// TwinCAT 3 PLC project tectrl
// ProgramVersion: 3.1.0.8
// libraries:
//   Tc2_Standard, * (Beckhoff Automation GmbH)
//   Tc2_System, * (Beckhoff Automation GmbH)
//   Tc3_Interfaces, * (Beckhoff Automation GmbH)
//   Tc3_Module, * (Beckhoff Automation GmbH)
//   Tc2_ControllerToolbox,3.4.1.0,Beckhoff Automation GmbH
//   Tc2_Math,3.3.0.0,Beckhoff Automation GmbH
//   Tc2_Utilities,3.3.8.0,Beckhoff Automation GmbH
//   Tc3_CM,newest,Beckhoff Automation GmbH
//   Tc3_MemMan,3.3.1.0,Beckhoff Automation GmbH
// project tree:
//   GVLs/ GVL.TcGVL
//   / PlcTask.TcTTO
//   POUs/components/ fb_ac_measurements.TcPOU, fb_discrete_pi.TcPOU, fb_flow_rate.TcPOU, fb_prod_feedforward.TcPOU, fb_ratio_trimming.TcPOU, fb_slewrate_limiter.TcPOU, fb_vel_pi.TcPOU (not stored), fb_xmeas_acquire.TcPOU (not stored), fb_unitdelay_real.TcPOU (not stored)
//   POUs/debug/ fb_generate_random_value.TcPOU (not stored), fb_xmeas_simulated.TcPOU (not stored)
//   POUs/ ldrMain.TcPOU
//   POUs/subsystems/ fb_ac_ratio_ctrl.TcPOU, fb_level_ctrl.TcPOU, fb_prod_rate_ctrl.TcPOU, fb_prod_comp_ctrl.TcPOU, fb_feed_ratio_ctrl.TcPOU (not stored), fb_temp_ctrl.TcPOU
//   POUs/test/ fb_test_xmeas_simulated.TcPOU (not stored)
// real-time tasks:
//   TASK PlcTask: cycle T#100000us, priority 20, ADS port 350

CONFIGURATION tectrl
    RESOURCE PLC ON TwinCAT3
        TASK PlcTask(INTERVAL := T#100000us, PRIORITY := 20);
        PROGRAM ldrMain WITH PlcTask : ldrMain;
    END_RESOURCE
END_CONFIGURATION

// ---- GVLs/GVL.TcGVL
VAR_GLOBAL
	
	// used for main start/stop/estop
	g_RUNNING: BOOL;
	g_START: BOOL;
	
	// E-STOP
	g_ESTOP: BOOL := TRUE;
	
	// loop control constants
	g_Ts_base : REAL := 0.001;
	g_Ts : REAL := 0.1;
	
	// the initial setpoints
	g_set_production: 		REAL := 22.89;
	g_set_stip_level: 		REAL := 50;
	g_set_sep_level:  		REAL := 50;
	g_set_reactor_level: 	REAL := 65;
	g_set_reactor_press: 	REAL := 2800;
	g_set_mol_pct_g:	 	REAL := 53.8;
	g_set_ya:				REAL := 100*32.2/(32.2+18.8);
	g_set_yac:				REAL := 32.2+18.8;
	g_set_reactor_temp:		REAL := 122.9;
	g_set_rcycle_valve_pos: REAL := 0;
	g_set_steam_valve_pos:	REAL := 0;
	g_set_agitator_speed:	REAL :=	100;		
	g_set_separator_temp:	REAL := SP17_0;
	
	// storage variables for sub-controllers
	g_xmeas: ARRAY [1..41] 	OF REAL;
	g_xmv: ARRAY [1..12] 	OF REAL := [50,50,65,2800,22.89,63.1373,51,122.9,0,0,100,53.8];
	g_rx: ARRAY [1..7] 		OF REAL;
	
	// production rate variables
	g_Prodsp: REAL;
	g_Fp: REAL;
	
	// Percent G Composition
	g_PctGsp: REAL;
	g_Eadj: REAL :=1.0;
	
	
	
END_VAR

VAR_GLOBAL CONSTANT
	Fp_0: REAL :=100;
	r_0 : ARRAY [1..7] OF REAL := 
		[0.251/Fp_0, 3664/Fp_0, 4509/Fp_0, 9.35/Fp_0, 0.337/Fp_0, 25.16/Fp_0, 22.95/Fp_0];    
              		
	xmv_0 : ARRAY [1..12] OF REAL := 
		[50,50,65,2800,22.89,63.1373,51,122.9,0,0,100,53.8];
	
	SP17_0 : REAL := 0.0;  // need value !!!
	Eadj_0 : REAL := 0.0;  // need value !!!
	ProdspGain: REAL := 100/22.89;	
END_VAR

// ---- POUs/ldrMain.TcPOU
PROGRAM ldrMain


// Notes
//  I imagine that the control loops can run as independent threads/tasks under the main PlcTask
//  xmeas, xmv, r, and maybe others could be stored in a GVL 
VAR
	
	// data acquitistion from IO blocks
	xmeas_acquire: fb_xmeas_acquire;

	// Molar Percent G control loop
	//pct_g_dpi: fb_discrete_pi		  := (kc:=1, ti:=0.001/60, Ts:=g_Ts_base, hi :=100, lo:=0, x0:=Eadj_0);
	
	// production rate control loop
	prod_rate_loop: fb_prod_rate_ctrl := (kc:=3.2, ti:=120/60, ts:=g_Ts_base, x0:=0, hi:=30, lo:=0);	
	
	// feed ratio control loop
	feed_ratio_ctrl: fb_feed_ratio_ctrl;
	
	// process levels/invetory controller
	level_ctrl: fb_level_ctrl;
		
	// product comnposition controller
	prod_comp_ctrl: fb_prod_comp_ctrl;
	
	// A & C ratio controller
	ac_ratio_ctrl: fb_ac_ratio_ctrl;
	
	// temperature controller
	temp_ctrl: fb_temp_ctrl;
	
END_VAR

VAR_INPUT
	
END_VAR
VAR // added by the converter: edge detectors and wires of the graphical bodies
    _w1 : BOOL;
END_VAR

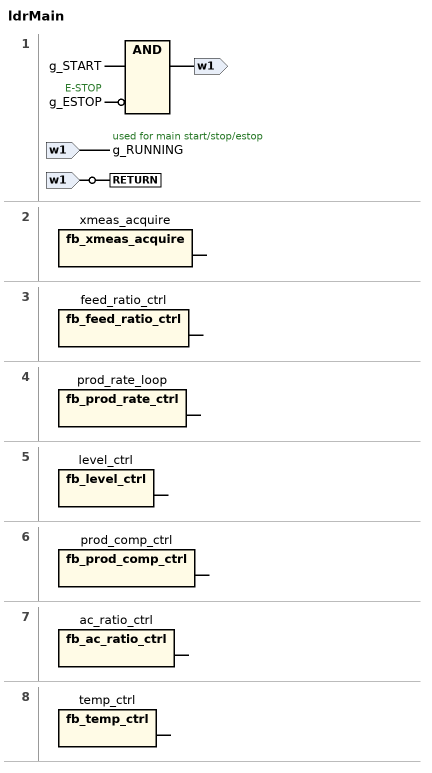
// NETWORK 1
//   g_ESTOP: E-STOP
//   g_RUNNING: used for main start/stop/estop
_w1 := g_START AND NOT g_ESTOP;
g_RUNNING := _w1;
IF NOT _w1 THEN RETURN; END_IF

// NETWORK 2
//   xmeas_acquire: data acquitistion from IO blocks
xmeas_acquire(); // fb_xmeas_acquire

// NETWORK 3
//   feed_ratio_ctrl: feed ratio control loop
feed_ratio_ctrl(); // fb_feed_ratio_ctrl

// NETWORK 4
//   prod_rate_loop: production rate control loop
prod_rate_loop(); // fb_prod_rate_ctrl

// NETWORK 5
//   level_ctrl: process levels/invetory controller
level_ctrl(); // fb_level_ctrl

// NETWORK 6
//   prod_comp_ctrl: product comnposition controller
prod_comp_ctrl(); // fb_prod_comp_ctrl

// NETWORK 7
//   ac_ratio_ctrl: A & C ratio controller
ac_ratio_ctrl(); // fb_ac_ratio_ctrl

// NETWORK 8
//   temp_ctrl: temperature controller
temp_ctrl(); // fb_temp_ctrl

END_PROGRAM

// ---- POUs/subsystems/fb_prod_rate_ctrl.TcPOU
FUNCTION_BLOCK fb_prod_rate_ctrl

VAR_INPUT
	kc: REAL;
	ti:REAL;
	ts:REAL;
	hi:REAL;
	lo:REAL;
	x0:REAL := 0;
	set_prod_rate: REAL := g_set_production;
	//xmv17: REAL;

END_VAR

VAR_OUTPUT
	Prodsp: REAL := 0;
	Fp: REAL :=0;
END_VAR

VAR
	
	vel_p: fb_vel_pi;
	x: FB_CTRL_2POINT;
	zoh_real_0: fb_zoh_real := (xlast := x0 );
	change_rate_limit: FB_CTRL_LIMITER := (stInternalParams := (fMinOutput := -0.286875, fMaxOutput := 0.286875));
	rate: REAL := 0;
	
	prodsp_scaled: REAL;
	calc_change_rate: FB_CTRL_D;
	integrate_change_rate: FB_CTRL_I;
	prod_rate_saturate: FB_CTRL_LIMITER;
	prod_rate_saturate_params: ST_CTRL_LIMITER_PARAMS := (fMinOutput := lo, fMaxOutput := hi);
	last_prod_rate: REAL := 0.0;
	
	stparams_calc_change_rate: ST_CTRL_D_PARAMS;
	stparams_change_rate_limit: ST_CTRL_LIMITER_PARAMS;
	stparams_integrate_change_rate: ST_CTRL_I_PARAMS;
	
END_VAR

VAR CONSTANT
	ProdspGain: REAL := 100/22.89;
END_VAR

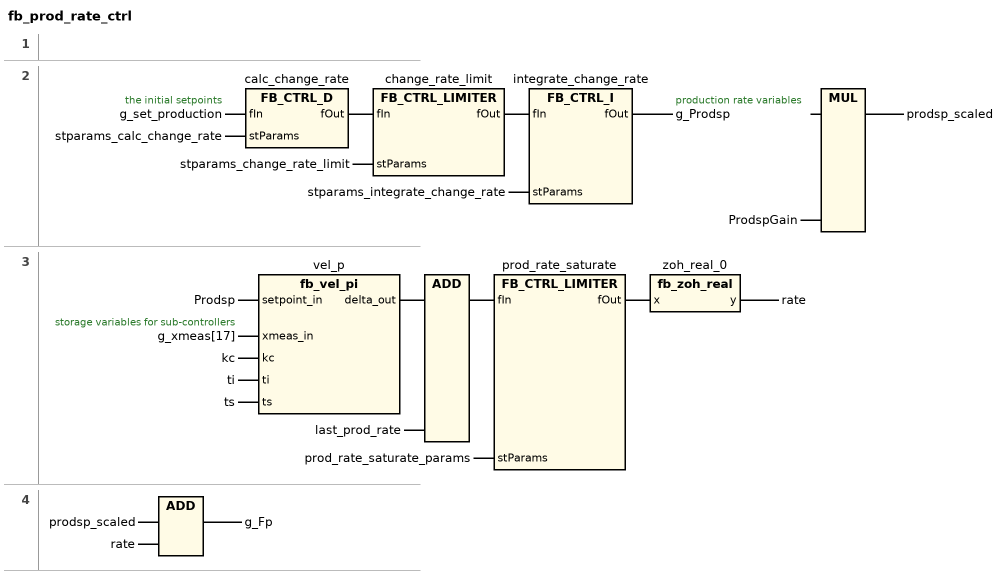
// NETWORK 1

// NETWORK 2
//   g_set_production: the initial setpoints
//   g_Prodsp: production rate variables
calc_change_rate(fIn := g_set_production, stParams := stparams_calc_change_rate); // FB_CTRL_D
change_rate_limit(fIn := calc_change_rate.fOut, stParams := stparams_change_rate_limit); // FB_CTRL_LIMITER
integrate_change_rate(fIn := change_rate_limit.fOut, stParams := stparams_integrate_change_rate); // FB_CTRL_I
g_Prodsp := integrate_change_rate.fOut;
prodsp_scaled := integrate_change_rate.fOut * ProdspGain;

// NETWORK 3
//   g_xmeas[17]: storage variables for sub-controllers
vel_p(setpoint_in := Prodsp, xmeas_in := g_xmeas[17], kc := kc, ti := ti, ts := ts); // fb_vel_pi
prod_rate_saturate(fIn := vel_p.delta_out + last_prod_rate, stParams := prod_rate_saturate_params); // FB_CTRL_LIMITER
zoh_real_0(x := prod_rate_saturate.fOut); // fb_zoh_real
rate := zoh_real_0.y;

// NETWORK 4
g_Fp := prodsp_scaled + rate;

END_FUNCTION_BLOCK

// ---- POUs/subsystems/fb_level_ctrl.TcPOU
FUNCTION_BLOCK fb_level_ctrl

VAR_INPUT
END_VAR

VAR_OUTPUT
END_VAR

VAR
	stripper_level_dpi: fb_discrete_pi			:= (kc:=2E-4, ti:=200/60, Ts:=g_Ts_base, hi :=100, lo:=0, x0:=r_0[7]);
	separator_level_dpi: fb_discrete_pi			:= (kc:=-1E-3, ti:=200/60, Ts:=g_Ts_base, hi :=100, lo:=0, x0:=r_0[6]);
	reactor_level_dpi: fb_discrete_pi			:= (kc:=0.8, ti:=60/60, Ts:=g_Ts_base, hi :=100, lo:=0, x0:=SP17_0);
	reactor_pressure_dpi: fb_discrete_pi		:= (kc:=-1E-4, ti:=20/60, Ts:=g_Ts_base, hi :=100, lo:=0, x0:=r_0[5]);
	reactor_temp_dpi: fb_discrete_pi			:= (kc:=-8, ti:=7.5/60, Ts:=g_Ts_base, hi :=100, lo:=0, x0:=xmv_0[10]);		
END_VAR

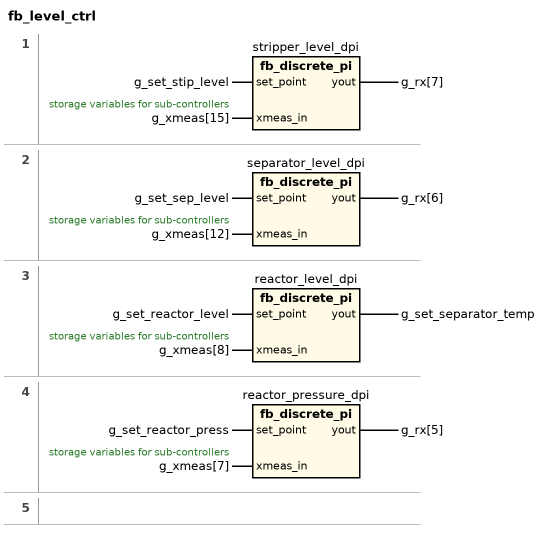
// NETWORK 1
//   g_xmeas[15]: storage variables for sub-controllers
stripper_level_dpi(set_point := g_set_stip_level, xmeas_in := g_xmeas[15]); // fb_discrete_pi
g_rx[7] := stripper_level_dpi.yout;

// NETWORK 2
//   g_xmeas[12]: storage variables for sub-controllers
separator_level_dpi(set_point := g_set_sep_level, xmeas_in := g_xmeas[12]); // fb_discrete_pi
g_rx[6] := separator_level_dpi.yout;

// NETWORK 3
//   g_xmeas[8]: storage variables for sub-controllers
reactor_level_dpi(set_point := g_set_reactor_level, xmeas_in := g_xmeas[8]); // fb_discrete_pi
g_set_separator_temp := reactor_level_dpi.yout;

// NETWORK 4
//   g_xmeas[7]: storage variables for sub-controllers
reactor_pressure_dpi(set_point := g_set_reactor_press, xmeas_in := g_xmeas[7]); // fb_discrete_pi
g_rx[5] := reactor_pressure_dpi.yout;

// NETWORK 5

END_FUNCTION_BLOCK

// ---- POUs/components/fb_discrete_pi.TcPOU
FUNCTION_BLOCK fb_discrete_pi

VAR_INPUT
	// signal inputs
	set_point: REAL := 0.0;
	xmeas_in: REAL := 0.0;
	
	// parameters
	kc: REAL;
	ti: REAL;
	ts: REAL;
	hi: REAL := 100;
	lo: REAL;
	x0: REAL;
		
END_VAR

VAR_OUTPUT
	yout: REAL; // needs to be initialized by caller
END_VAR

VAR
	vel_pi: fb_vel_pi := (kc:=kc, ti:=ti, ts:=ts);
	dpi_unit_delay: fb_unitdelay_real := (xlast:=x0);
END_VAR

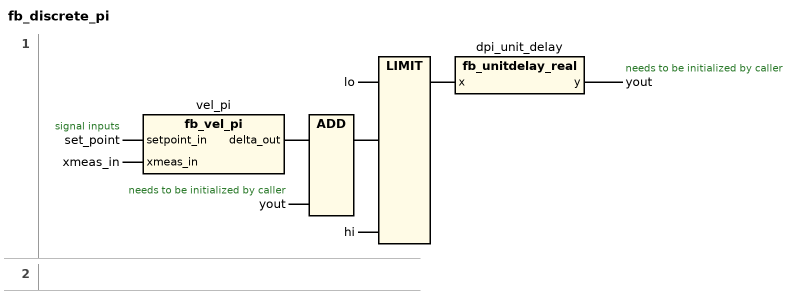
// NETWORK 1
//   set_point: signal inputs
//   yout: needs to be initialized by caller
vel_pi(setpoint_in := set_point, xmeas_in := xmeas_in); // fb_vel_pi
dpi_unit_delay(x := LIMIT(lo, vel_pi.delta_out + yout, hi)); // fb_unitdelay_real
yout := dpi_unit_delay.y;

// NETWORK 2

END_FUNCTION_BLOCK

// ---- POUs/subsystems/fb_prod_comp_ctrl.TcPOU
FUNCTION_BLOCK fb_prod_comp_ctrl

VAR_INPUT
	kc: REAL := 0.0;
	ti:REAL := 0.0;
	ts:REAL := 0.0;
	hi:REAL := 0.0;
	lo:REAL := 0.0;
	x0:REAL := 0.0;
	set_prod_rate: REAL := g_set_production;
	//xmv17: REAL;

END_VAR

VAR_OUTPUT
	Prodsp: REAL := 0;
	Fp: REAL :=0;
END_VAR

VAR
	
	pct_g_dpi: fb_discrete_pi := (kc := 0.4, ti := 100.0, ts := g_Ts_base, hi := 100, lo:=0.0);
	zoh_real_0: fb_zoh_real := (xlast := x0 );
	change_rate_limit: FB_CTRL_LIMITER := (stInternalParams := (fMinOutput := -0.286875, fMaxOutput := 0.286875));
	rate: REAL := 0;
	
	prodsp_scaled: REAL;
	calc_change_rate: FB_CTRL_D;
	integrate_change_rate: FB_CTRL_I;
	prod_rate_saturate: FB_CTRL_LIMITER;
	prod_rate_saturate_params: ST_CTRL_LIMITER_PARAMS := (fMinOutput := lo, fMaxOutput := hi);
	last_prod_rate: REAL := 0.0;
	
	stparams_calc_change_rate: ST_CTRL_D_PARAMS;
	stparams_change_rate_limit: ST_CTRL_LIMITER_PARAMS;
	stparams_integrate_change_rate: ST_CTRL_I_PARAMS;
	
	pctgsp: REAL := 0.0;
	
	
	prod_feedforward: fb_prod_feedforward;
END_VAR

VAR CONSTANT
	ProdspGain: REAL := 100/22.89;
END_VAR

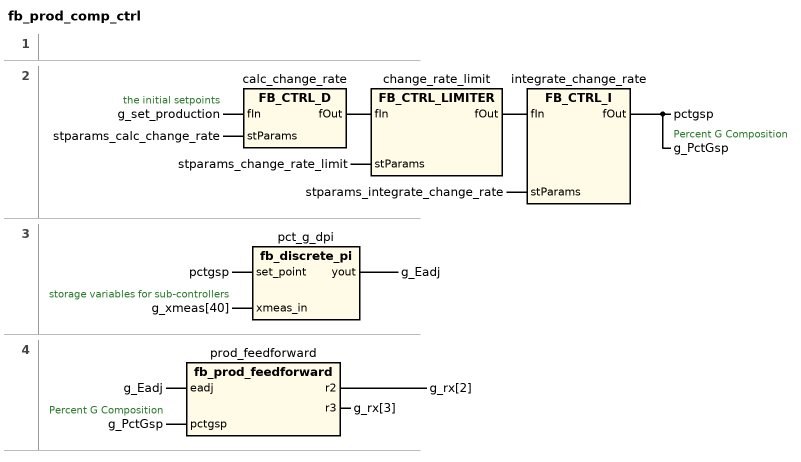
// NETWORK 1

// NETWORK 2
//   g_set_production: the initial setpoints
//   g_PctGsp: Percent G Composition
calc_change_rate(fIn := g_set_production, stParams := stparams_calc_change_rate); // FB_CTRL_D
change_rate_limit(fIn := calc_change_rate.fOut, stParams := stparams_change_rate_limit); // FB_CTRL_LIMITER
integrate_change_rate(fIn := change_rate_limit.fOut, stParams := stparams_integrate_change_rate); // FB_CTRL_I
pctgsp := integrate_change_rate.fOut;
g_PctGsp := integrate_change_rate.fOut;

// NETWORK 3
//   g_xmeas[40]: storage variables for sub-controllers
pct_g_dpi(set_point := pctgsp, xmeas_in := g_xmeas[40]); // fb_discrete_pi
g_Eadj := pct_g_dpi.yout;

// NETWORK 4
//   g_PctGsp: Percent G Composition
prod_feedforward(eadj := g_Eadj, pctgsp := g_PctGsp, r3 => g_rx[3]); // fb_prod_feedforward
g_rx[2] := prod_feedforward.r2;

END_FUNCTION_BLOCK

// ---- POUs/components/fb_prod_feedforward.TcPOU
FUNCTION_BLOCK fb_prod_feedforward

VAR_INPUT	
	eadj: REAL;
	pctgsp: REAL;
END_VAR

VAR_OUTPUT
	r2: REAL;
	r3: REAL;
END_VAR

VAR
	pctgspP2: REAL;
	pctgspP3: REAL;
	eadjProd1: REAL;
	eadjProd2: REAL;
END_VAR

VAR CONSTANT
	P2: ARRAY[0..2] OF REAL := [1.5192E-3, 5.9446E-1, 2.7690E-1]; 
	P3: ARRAY[0..2] OF REAL := [-1.1377E-3, -8.0893E-1, 9.1060E1]; 
END_VAR


pctgspP2 := P2[0]*EXPT(pctgsp,2) + P2[1]*pctgsp + P2[2];
pctgspP3 := P2[0]*EXPT(pctgsp,2) + P2[1]*pctgsp + P2[2];
g_rx[2] :=  pctgspP2 - (32*eadj)/g_Fp;
g_rx[3] :=  pctgspP2 + (46*eadj)/g_Fp;

END_FUNCTION_BLOCK

// ---- POUs/subsystems/fb_ac_ratio_ctrl.TcPOU
FUNCTION_BLOCK fb_ac_ratio_ctrl

VAR_INPUT
	(*
	set_ya:  REAL := g_set_ya;
	set_yac: REAL := g_set_yac;
	xmeas11: REAL := g_xmeas[11];
	xmeas23: REAL := g_xmeas[23];
	xmeas25: REAL := g_xmeas[25];
	*)
END_VAR

VAR_OUTPUT
END_VAR

VAR
	// A & C measurements
	yA: 	REAL;
	yAC:	REAL;
	
	// yA control looop
	ya_control: fb_vel_pi := (kc := 0.0002, ti := 1.0, ts := g_Ts);
	ya_control_kc :	REAL := 0.0;
	loop14:	REAL := 0.0;
	
	// yAC control loop
	yac_control: fb_vel_pi := (kc := 0.0003, ti := 2, ts := g_Ts);
	loop15: REAL := 0.0;	
	
	// ratio trimming
	ratio_trimming: fb_ratio_trimming;
	
	// fine ac adjustments
	ac_measurements: fb_ac_measurements;
	separator_temp_dpi: fb_discrete_pi		:= (kc:=-4, ti:=15/60, Ts:=g_Ts_base, hi :=100, lo:=0, yout:=xmv_0[11]);	
	ratio_trimming_0: fb_ratio_trimming 	:= (r1 := g_rx[1], r4 := g_rx[4]);

END_VAR

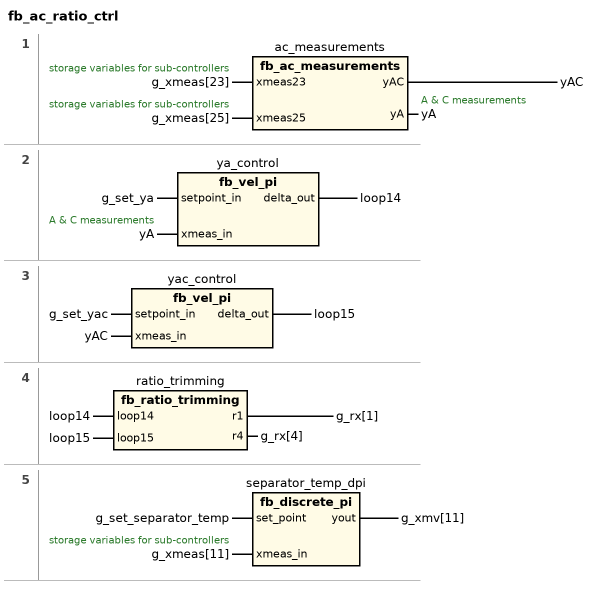
// NETWORK 1
//   ac_measurements: fine ac adjustments
//   g_xmeas[23]: storage variables for sub-controllers
//   g_xmeas[25]: storage variables for sub-controllers
//   yA: A & C measurements
ac_measurements(xmeas23 := g_xmeas[23], xmeas25 := g_xmeas[25], yA => yA); // fb_ac_measurements
yAC := ac_measurements.yAC;

// NETWORK 2
//   ya_control: yA control looop
//   yA: A & C measurements
ya_control(setpoint_in := g_set_ya, xmeas_in := yA); // fb_vel_pi
loop14 := ya_control.delta_out;

// NETWORK 3
//   yac_control: yAC control loop
yac_control(setpoint_in := g_set_yac, xmeas_in := yAC); // fb_vel_pi
loop15 := yac_control.delta_out;

// NETWORK 4
//   ratio_trimming: ratio trimming
ratio_trimming(loop14 := loop14, loop15 := loop15, r4 => g_rx[4]); // fb_ratio_trimming
g_rx[1] := ratio_trimming.r1;

// NETWORK 5
//   g_xmeas[11]: storage variables for sub-controllers
separator_temp_dpi(set_point := g_set_separator_temp, xmeas_in := g_xmeas[11]); // fb_discrete_pi
g_xmv[11] := separator_temp_dpi.yout;

END_FUNCTION_BLOCK

// ---- POUs/components/fb_ratio_trimming.TcPOU
FUNCTION_BLOCK fb_ratio_trimming

VAR_INPUT
	loop14: REAL;
	loop15: REAL;
END_VAR

VAR_OUTPUT
	r1: REAL;
	r4: REAL;
END_VAR

VAR
END_VAR


r1 := loop14 + r1;
r4 := loop15 - loop14 + r4;

END_FUNCTION_BLOCK

// ---- POUs/components/fb_ac_measurements.TcPOU
FUNCTION_BLOCK fb_ac_measurements

VAR_INPUT
	xmeas23 : REAL := 0.0;
	xmeas25 : REAL := 0.0;
END_VAR

VAR_OUTPUT
	yAC : REAL := 0.0;
	yA : REAL := 0.0;
	
	
END_VAR

VAR
END_VAR


yAC := xmeas23 + xmeas25;
yA := xmeas23*100/yAC;

END_FUNCTION_BLOCK

// ---- POUs/subsystems/fb_temp_ctrl.TcPOU
FUNCTION_BLOCK fb_temp_ctrl

VAR_INPUT
END_VAR

VAR_OUTPUT	
END_VAR

VAR
	separator_temp_dpi: fb_discrete_pi		:= (kc:=-4, ti:=15/60, Ts:=g_Ts_base, hi :=100, lo:=0, yout:=xmv_0[11]);	
	reactor_temp_dpi: fb_discrete_pi		:= (kc:=-8, ti:=7.5/60, Ts:=g_Ts_base, hi :=100, lo:=0, yout:=xmv_0[10]);
	
END_VAR

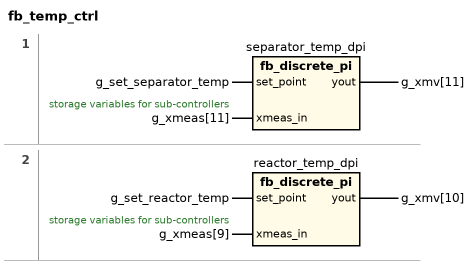
// NETWORK 1
//   g_xmeas[11]: storage variables for sub-controllers
separator_temp_dpi(set_point := g_set_separator_temp, xmeas_in := g_xmeas[11]); // fb_discrete_pi
g_xmv[11] := separator_temp_dpi.yout;

// NETWORK 2
//   g_xmeas[9]: storage variables for sub-controllers
reactor_temp_dpi(set_point := g_set_reactor_temp, xmeas_in := g_xmeas[9]); // fb_discrete_pi
g_xmv[10] := reactor_temp_dpi.yout;

END_FUNCTION_BLOCK

// ---- POUs/components/fb_flow_rate.TcPOU
FUNCTION_BLOCK fb_flow_rate

VAR_INPUT
	// signal inputs
	ratio_in: REAL := 0.0;
	xmeas_in: REAL := 0.0;
	
	// parameters
	kc: REAL := 0.0;
	ti: REAL := 0.0;
	ts: REAL := 0.0;
	hi: REAL := 2E32;
	lo: REAL := 0;
	
END_VAR

VAR_OUTPUT
	yout: REAL; // needs to be initialized by caller
END_VAR

VAR
	vel_pi: fb_vel_pi;
END_VAR

END_FUNCTION_BLOCK

// ---- POUs/components/fb_slewrate_limiter.TcPOU
FUNCTION_BLOCK fb_slewrate_limiter

VAR_INPUT
	in: REAL;
	pos_slewrate_limit: REAL := 0.0;
	neg_slewrate_limit: REAL := 0.0;
END_VAR

VAR_OUTPUT
	out: REAL;
END_VAR

VAR
	
	last_in: REAL := g_set_production;
	slope: REAL;

	fbCTRL_GET_TASK_CYCLETIME   : FB_CTRL_GET_TASK_CYCLETIME;
	tTaskCycleTime: TIME;
	bCycleTimeValid: BOOL;
	eErrorId: TC2_CONTROLLERTOOLBOX.E_CTRL_ERRORCODES;
	bError: BOOL;
    eState: E_CTRL_STATE;

END_VAR


fbCTRL_GET_TASK_CYCLETIME( eMode:=eCTRL_MODE_ACTIVE, tTaskCycleTime=>tTaskCycleTime, 
	bCycleTimeValid => bCycleTimeValid, 
	eState 			=> eState,
	eErrorId        => eErrorId,
    bError          => bError); 

IF bCycleTimevalid THEN 
	tTaskCycleTime :=fbCTRL_GET_TASK_CYCLETIME.tTaskCycleTime;
	
	slope := (last_in - in)/TIME_TO_REAL(tTaskCycleTime);
	IF slope >= pos_slewrate_limit THEN
		out := last_in + pos_slewrate_limit;
	ELSIF slope > pos_slewrate_limit THEN
		out := last_in - neg_slewrate_limit;
	ELSE
		out := in;	
	END_IF
ELSE
	out := last_in;
END_IF
last_in := in;

END_FUNCTION_BLOCK
